KUKA KRL program: redrabbit.src, RedRabbit.dat

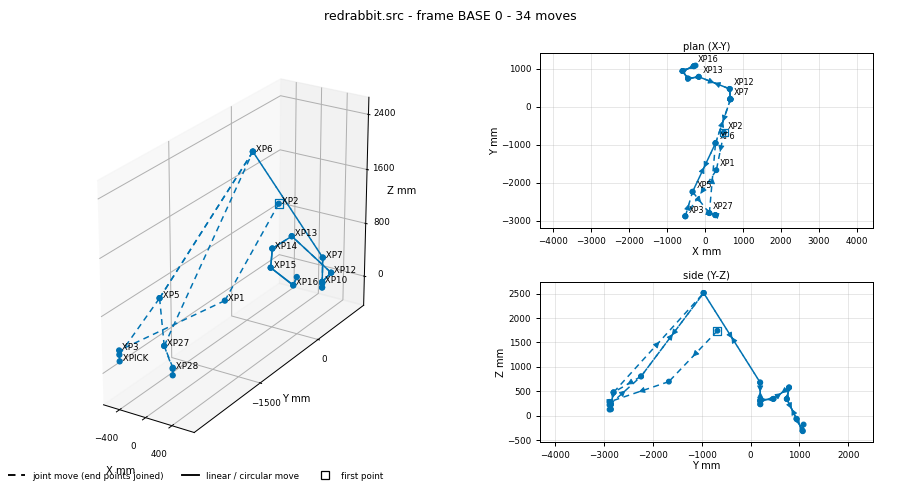
[picture p0: tool path of redrabbit.src in frame BASE 0, 34 of 36 moves have a stored position in this frame; points joined in program order, loops and branches not executed]
--- redrabbit.src ---
&ACCESS RVO1
&REL 74
&PARAM EDITMASK = *
&PARAM TEMPLATE = C:\KRC\TP\Nutweld\Template\NutWeld_Vorgabe
DEF RedRabbit( )
;FOLD INI
  ;FOLD BASISTECH INI
    GLOBAL INTERRUPT DECL 3 WHEN $STOPMESS==TRUE DO IR_STOPM ( )
    INTERRUPT ON 3
    BAS (#INITMOV,0 )
  ;ENDFOLD (BASISTECH INI)
	;FOLD NutWeld
	;ENDFOLD (NutWeld)
  ;FOLD USER INI
    ;Make your modifications here
do141Spare=FALSE
do142Spare=FALSE
  ;ENDFOLD (USER INI)
;ENDFOLD (INI)
wait for false

;FOLD PTP HOME  Vel= 100 % DEFAULT;%{PE}%MKUKATPBASIS,%CMOVE,%VPTP,%P 1:PTP, 2:HOME, 3:, 5:100, 7:DEFAULT
$BWDSTART = FALSE
PDAT_ACT=PDEFAULT
FDAT_ACT=FHOME
BAS (#PTP_PARAMS,100 )
$H_POS=XHOME
PTP  XHOME
;ENDFOLD
;FOLD Gripper SET [1]Gripper1 State=[1]OPEN Wait 0.2[s] Check with Strategy 1 ;%{PE}
;FOLD Parameters Parameters ;%{h}
;Params IlfProvider=GripperTech.GripperSet;setgripper=1;setstate=1;setcont=nocont;waittime=0.2;errorstrategy=1
;ENDFOLD
GRPg_SetStateAndCheck(1, 1, 0.2, 1)
;ENDFOLD
;FOLD Gripper SET [2]Gripper2 State=[2]CLOSE Wait 0.2[s] Check with Strategy 1 ;%{PE}
;FOLD Parameters Parameters ;%{h}
;Params IlfProvider=GripperTech.GripperSet;setgripper=2;setstate=2;setcont=nocont;waittime=0.2;errorstrategy=1
;ENDFOLD
GRPg_SetStateAndCheck(2, 2, 0.2, 1)
;ENDFOLD
;FOLD Gripper SET [3]Gripper3 State=[1]OPEN Wait 0.2[s] Check with Strategy 1 ;%{PE}
;FOLD Parameters Parameters ;%{h}
;Params IlfProvider=GripperTech.GripperSet;setgripper=3;setstate=1;setcont=nocont;waittime=0.2;errorstrategy=1
;ENDFOLD
GRPg_SetStateAndCheck(3, 1, 0.2, 1)
;ENDFOLD
;FOLD Gripper SET [4]Gripper4 State=[2]CLOSE Wait 0.2[s] Check with Strategy 1 ;%{PE}
;FOLD Parameters Parameters ;%{h}
;Params IlfProvider=GripperTech.GripperSet;setgripper=4;setstate=2;setcont=nocont;waittime=0.2;errorstrategy=1
;ENDFOLD
GRPg_SetStateAndCheck(4, 2, 0.2, 1)
;ENDFOLD
;FOLD PTP P2 Vel=100 % PDAT2 Tool[1]:TOOL 1 Base[0];%{PE}%R 8.3.43,%MKUKATPBASIS,%CMOVE,%VPTP,%P 1:PTP, 2:P2, 3:, 5:100, 7:PDAT2
$BWDSTART=FALSE
PDAT_ACT=PPDAT2
FDAT_ACT=FP2
BAS(#PTP_PARAMS,100)
PTP XP2
;ENDFOLD
;FOLD PTP P1 Vel=100 % PDAT1 Tool[1]:TOOL 1 Base[0];%{PE}%R 8.3.43,%MKUKATPBASIS,%CMOVE,%VPTP,%P 1:PTP, 2:P1, 3:, 5:100, 7:PDAT1
$BWDSTART=FALSE
PDAT_ACT=PPDAT1
FDAT_ACT=FP1
BAS(#PTP_PARAMS,100)
PTP XP1
;ENDFOLD
;FOLD PTP P3 Vel=100 % PDAT3 Tool[2]:TOOL 2 Base[0];%{PE}%R 8.3.43,%MKUKATPBASIS,%CMOVE,%VPTP,%P 1:PTP, 2:P3, 3:, 5:100, 7:PDAT3
$BWDSTART=FALSE
PDAT_ACT=PPDAT3
FDAT_ACT=FP3
BAS(#PTP_PARAMS,100)
PTP XP3
;ENDFOLD
;FOLD LIN PICK Vel=1 m/s CPDAT1 Tool[2]:TOOL 2 Base[0];%{PE}%R 8.3.43,%MKUKATPBASIS,%CMOVE,%VLIN,%P 1:LIN, 2:PICK, 3:, 5:1, 7:CPDAT1
$BWDSTART=FALSE
LDAT_ACT=LCPDAT1
FDAT_ACT=FPICK
BAS(#CP_PARAMS,1)
LIN XPICK
;ENDFOLD
;FOLD Gripper SET [3]Gripper3 State=[2]CLOSE Wait 0.2[s] Check with Strategy 1 ;%{PE}
;FOLD Parameters Parameters ;%{h}
;Params IlfProvider=GripperTech.GripperSet;setgripper=3;setstate=2;setcont=nocont;waittime=0.2;errorstrategy=1
;ENDFOLD
GRPg_SetStateAndCheck(3, 2, 0.2, 1)
;ENDFOLD
;FOLD Gripper CHECK [3]Gripper3 State=[2]CLOSE with Strategy 1 ;%{PE}
;FOLD Parameters Parameters ;%{h}
;Params IlfProvider=GripperTech.GripperCheck;setgripper=3;setstate=2;setcont=nocont;checkstrategy=1
;ENDFOLD
GRPg_Check(3, 2, FALSE, 1)
;ENDFOLD
;FOLD LIN P4 Vel=1 m/s CPDAT2 Tool[2]:TOOL 2 Base[0];%{PE}%R 8.3.43,%MKUKATPBASIS,%CMOVE,%VLIN,%P 1:LIN, 2:P4, 3:, 5:1, 7:CPDAT2
$BWDSTART=FALSE
LDAT_ACT=LCPDAT2
FDAT_ACT=FP4
BAS(#CP_PARAMS,1)
LIN XP4
;ENDFOLD
;FOLD PTP P5 Vel=100 % PDAT4 Tool[2]:TOOL 2 Base[0];%{PE}%R 8.3.43,%MKUKATPBASIS,%CMOVE,%VPTP,%P 1:PTP, 2:P5, 3:, 5:100, 7:PDAT4
$BWDSTART=FALSE
PDAT_ACT=PPDAT4
FDAT_ACT=FP5
BAS(#PTP_PARAMS,100)
PTP XP5
;ENDFOLD
;FOLD PTP P6 Vel=100 % PDAT5 Tool[2]:TOOL 2 Base[0];%{PE}%R 8.3.43,%MKUKATPBASIS,%CMOVE,%VPTP,%P 1:PTP, 2:P6, 3:, 5:100, 7:PDAT5
$BWDSTART=FALSE
PDAT_ACT=PPDAT5
FDAT_ACT=FP6
BAS(#PTP_PARAMS,100)
PTP XP6
;ENDFOLD
;Pick RH RedRabbit
;FOLD OUT 120 'do120Spare' State=TRUE ;%{PE}%R 8.3.43,%MKUKATPBASIS,%COUT,%VOUTX,%P 2:120, 3:do120Spare, 5:TRUE, 6:
$OUT[120]=TRUE
;ENDFOLD
;FOLD WAIT FOR ( IN 98 'di098Spare' );%{PE}%R 8.3.43,%MKUKATPBASIS,%CEXT_WAIT_FOR,%VEXT_WAIT_FOR,%P 2:, 4:, 5:$IN, 6:98, 7:di098Spare, 9:
WAIT FOR  ( $IN[98] )
;ENDFOLD
;FOLD PTP P7 Vel=100 % PDAT9 Tool[2]:TOOL 2 Base[0];%{PE}%R 8.3.43,%MKUKATPBASIS,%CMOVE,%VPTP,%P 1:PTP, 2:P7, 3:, 5:100, 7:PDAT9
$BWDSTART=FALSE
PDAT_ACT=PPDAT9
FDAT_ACT=FP7
BAS(#PTP_PARAMS,100)
PTP XP7
;ENDFOLD
;FOLD LIN P10 Vel=1 m/s CPDAT4 Tool[2]:TOOL 2 Base[0];%{PE}%R 8.3.43,%MKUKATPBASIS,%CMOVE,%VLIN,%P 1:LIN, 2:P10, 3:, 5:1, 7:CPDAT4
$BWDSTART=FALSE
LDAT_ACT=LCPDAT4
FDAT_ACT=FP10
BAS(#CP_PARAMS,1)
LIN XP10
;ENDFOLD
;FOLD LIN PICK2 Vel=1 m/s CPDAT5 Tool[2]:TOOL 2 Base[0];%{PE}%R 8.3.43,%MKUKATPBASIS,%CMOVE,%VLIN,%P 1:LIN, 2:PICK2, 3:, 5:1, 7:CPDAT5
$BWDSTART=FALSE
LDAT_ACT=LCPDAT5
FDAT_ACT=FPICK2
BAS(#CP_PARAMS,1)
LIN XPICK2
;ENDFOLD
;FOLD Gripper SET [1]Gripper1 State=[2]CLOSE Wait 0.2[s] Check with Strategy 1 ;%{PE}
;FOLD Parameters Parameters ;%{h}
;Params IlfProvider=GripperTech.GripperSet;setgripper=1;setstate=2;setcont=nocont;waittime=0.2;errorstrategy=1
;ENDFOLD
GRPg_SetStateAndCheck(1, 2, 0.2, 1)
;ENDFOLD
;FOLD Gripper CHECK [1]Gripper1 State=[2]CLOSE with Strategy 1 ;%{PE}
;FOLD Parameters Parameters ;%{h}
;Params IlfProvider=GripperTech.GripperCheck;setgripper=1;setstate=2;setcont=nocont;checkstrategy=1
;ENDFOLD
GRPg_Check(1, 2, FALSE, 1)
;ENDFOLD
;FOLD LIN P11 Vel=1 m/s CPDAT6 Tool[2]:TOOL 2 Base[0];%{PE}%R 8.3.43,%MKUKATPBASIS,%CMOVE,%VLIN,%P 1:LIN, 2:P11, 3:, 5:1, 7:CPDAT6
$BWDSTART=FALSE
LDAT_ACT=LCPDAT6
FDAT_ACT=FP11
BAS(#CP_PARAMS,1)
LIN XP11
;ENDFOLD
;FOLD LIN P12 Vel=1 m/s CPDAT7 Tool[2]:TOOL 2 Base[0];%{PE}%R 8.3.43,%MKUKATPBASIS,%CMOVE,%VLIN,%P 1:LIN, 2:P12, 3:, 5:1, 7:CPDAT7
$BWDSTART=FALSE
LDAT_ACT=LCPDAT7
FDAT_ACT=FP12
BAS(#CP_PARAMS,1)
LIN XP12
;ENDFOLD
;FOLD PTP P13 Vel=100 % PDAT10 Tool[2]:TOOL 2 Base[0];%{PE}%R 8.3.43,%MKUKATPBASIS,%CMOVE,%VPTP,%P 1:PTP, 2:P13, 3:, 5:100, 7:PDAT10
$BWDSTART=FALSE
PDAT_ACT=PPDAT10
FDAT_ACT=FP13
BAS(#PTP_PARAMS,100)
PTP XP13
;ENDFOLD
;FOLD LIN P14 Vel=1 m/s CPDAT8 Tool[2]:TOOL 2 Base[0];%{PE}%R 8.3.43,%MKUKATPBASIS,%CMOVE,%VLIN,%P 1:LIN, 2:P14, 3:, 5:1, 7:CPDAT8
$BWDSTART=FALSE
LDAT_ACT=LCPDAT8
FDAT_ACT=FP14
BAS(#CP_PARAMS,1)
LIN XP14
;ENDFOLD
;FOLD LIN P15 Vel=1 m/s CPDAT9 Tool[2]:TOOL 2 Base[0];%{PE}%R 8.3.43,%MKUKATPBASIS,%CMOVE,%VLIN,%P 1:LIN, 2:P15, 3:, 5:1, 7:CPDAT9
$BWDSTART=FALSE
LDAT_ACT=LCPDAT9
FDAT_ACT=FP15
BAS(#CP_PARAMS,1)
LIN XP15
;ENDFOLD
;FOLD LIN P16 Vel=1 m/s CPDAT10 Tool[2]:TOOL 2 Base[0];%{PE}%R 8.3.43,%MKUKATPBASIS,%CMOVE,%VLIN,%P 1:LIN, 2:P16, 3:, 5:1, 7:CPDAT10
$BWDSTART=FALSE
LDAT_ACT=LCPDAT10
FDAT_ACT=FP16
BAS(#CP_PARAMS,1)
LIN XP16
;ENDFOLD
;FOLD LIN NUTCHECK Vel=1 m/s CPDAT11 Tool[2]:TOOL 2 Base[0];%{PE}%R 8.3.43,%MKUKATPBASIS,%CMOVE,%VLIN,%P 1:LIN, 2:NUTCHECK, 3:, 5:1, 7:CPDAT11
$BWDSTART=FALSE
LDAT_ACT=LCPDAT11
FDAT_ACT=FNUTCHECK
BAS(#CP_PARAMS,1)
LIN XNUTCHECK
;ENDFOLD
;FOLD WAIT Time=1 sec;%{PE}%R 8.3.43,%MKUKATPBASIS,%CWAIT,%VWAIT,%P 3:1
WAIT SEC 1
;ENDFOLD
IF ((di777StudPartPresent1==FALSE) AND (di778StudPartPresent2==FALSE) AND (di779StudPartPresent3==FALSE) AND (di780StudPartPresent4==FALSE) AND (Di781StudPartPresent5==FALSE) AND (di782StudPartPresent6==FALSE)) THEN
do142Spare=TRUE
ELSE
do141Spare=TRUE
ENDIF
;FOLD PTP P17 Vel=100 % PDAT11 Tool[2]:TOOL 2 Base[0];%{PE}%R 8.3.43,%MKUKATPBASIS,%CMOVE,%VPTP,%P 1:PTP, 2:P17, 3:, 5:100, 7:PDAT11
$BWDSTART=FALSE
PDAT_ACT=PPDAT11
FDAT_ACT=FP17
BAS(#PTP_PARAMS,100)
PTP XP17
;ENDFOLD
;FOLD LIN P18 Vel=1 m/s CPDAT12 Tool[2]:TOOL 2 Base[0];%{PE}%R 8.3.43,%MKUKATPBASIS,%CMOVE,%VLIN,%P 1:LIN, 2:P18, 3:, 5:1, 7:CPDAT12
$BWDSTART=FALSE
LDAT_ACT=LCPDAT12
FDAT_ACT=FP18
BAS(#CP_PARAMS,1)
LIN XP18
;ENDFOLD
;FOLD LIN P19 Vel=1 m/s CPDAT13 Tool[2]:TOOL 2 Base[0];%{PE}%R 8.3.43,%MKUKATPBASIS,%CMOVE,%VLIN,%P 1:LIN, 2:P19, 3:, 5:1, 7:CPDAT13
$BWDSTART=FALSE
LDAT_ACT=LCPDAT13
FDAT_ACT=FP19
BAS(#CP_PARAMS,1)
LIN XP19
;ENDFOLD
;FOLD PTP P20 Vel=100 % PDAT12 Tool[2]:TOOL 2 Base[0];%{PE}%R 8.3.43,%MKUKATPBASIS,%CMOVE,%VPTP,%P 1:PTP, 2:P20, 3:, 5:100, 7:PDAT12
$BWDSTART=FALSE
PDAT_ACT=PPDAT12
FDAT_ACT=FP20
BAS(#PTP_PARAMS,100)
PTP XP20
;ENDFOLD
;FOLD LIN P21 Vel=1 m/s CPDAT14 Tool[2]:TOOL 2 Base[0];%{PE}%R 8.3.43,%MKUKATPBASIS,%CMOVE,%VLIN,%P 1:LIN, 2:P21, 3:, 5:1, 7:CPDAT14
$BWDSTART=FALSE
LDAT_ACT=LCPDAT14
FDAT_ACT=FP21
BAS(#CP_PARAMS,1)
LIN XP21
;ENDFOLD
;FOLD LIN P22 Vel=1 m/s CPDAT15 Tool[2]:TOOL 2 Base[0];%{PE}%R 8.3.43,%MKUKATPBASIS,%CMOVE,%VLIN,%P 1:LIN, 2:P22, 3:, 5:1, 7:CPDAT15
$BWDSTART=FALSE
LDAT_ACT=LCPDAT15
FDAT_ACT=FP22
BAS(#CP_PARAMS,1)
LIN XP22
;ENDFOLD
;FOLD LIN DROP Vel=1 m/s CPDAT16 Tool[2]:TOOL 2 Base[0];%{PE}%R 8.3.43,%MKUKATPBASIS,%CMOVE,%VLIN,%P 1:LIN, 2:DROP, 3:, 5:1, 7:CPDAT16
$BWDSTART=FALSE
LDAT_ACT=LCPDAT16
FDAT_ACT=FDROP
BAS(#CP_PARAMS,1)
LIN XDROP
;ENDFOLD
;FOLD Gripper SET [2]Gripper2 State=[1]OPEN Wait 0.2[s] Check with Strategy 1 ;%{PE}
;FOLD Parameters Parameters ;%{h}
;Params IlfProvider=GripperTech.GripperSet;setgripper=2;setstate=1;setcont=nocont;waittime=0.2;errorstrategy=1
;ENDFOLD
GRPg_SetStateAndCheck(2, 1, 0.2, 1)
;ENDFOLD
;FOLD Gripper SET [1]Gripper1 State=[1]OPEN Wait 0.2[s] Check with Strategy 1 ;%{PE}
;FOLD Parameters Parameters ;%{h}
;Params IlfProvider=GripperTech.GripperSet;setgripper=1;setstate=1;setcont=nocont;waittime=0.2;errorstrategy=1
;ENDFOLD
GRPg_SetStateAndCheck(1, 1, 0.2, 1)
;ENDFOLD
;FOLD Gripper CHECK [2]Gripper2 State=[1]OPEN with Strategy 1 ;%{PE}
;FOLD Parameters Parameters ;%{h}
;Params IlfProvider=GripperTech.GripperCheck;setgripper=2;setstate=1;setcont=nocont;checkstrategy=1
;ENDFOLD
GRPg_Check(2, 1, FALSE, 1)
;ENDFOLD
;FOLD Gripper CHECK [1]Gripper1 State=[1]OPEN with Strategy 1 ;%{PE}
;FOLD Parameters Parameters ;%{h}
;Params IlfProvider=GripperTech.GripperCheck;setgripper=1;setstate=1;setcont=nocont;checkstrategy=1
;ENDFOLD
GRPg_Check(1, 1, FALSE, 1)
;ENDFOLD
;FOLD LIN P23 Vel=1 m/s CPDAT17 Tool[2]:TOOL 2 Base[0];%{PE}%R 8.3.43,%MKUKATPBASIS,%CMOVE,%VLIN,%P 1:LIN, 2:P23, 3:, 5:1, 7:CPDAT17
$BWDSTART=FALSE
LDAT_ACT=LCPDAT17
FDAT_ACT=FP23
BAS(#CP_PARAMS,1)
LIN XP23
;ENDFOLD
;FOLD PTP P24 Vel=100 % PDAT13 Tool[2]:TOOL 2 Base[0];%{PE}%R 8.3.43,%MKUKATPBASIS,%CMOVE,%VPTP,%P 1:PTP, 2:P24, 3:, 5:100, 7:PDAT13
$BWDSTART=FALSE
PDAT_ACT=PPDAT13
FDAT_ACT=FP24
BAS(#PTP_PARAMS,100)
PTP XP24
;ENDFOLD
;FOLD PTP P25 Vel=100 % PDAT14 Tool[2]:TOOL 2 Base[0];%{PE}%R 8.3.43,%MKUKATPBASIS,%CMOVE,%VPTP,%P 1:PTP, 2:P25, 3:, 5:100, 7:PDAT14
$BWDSTART=FALSE
PDAT_ACT=PPDAT14
FDAT_ACT=FP25
BAS(#PTP_PARAMS,100)
PTP XP25
;ENDFOLD
;FOLD OUT 120 'do120Spare' State=FALSE ;%{PE}%R 8.3.43,%MKUKATPBASIS,%COUT,%VOUTX,%P 2:120, 3:do120Spare, 5:FALSE, 6:
$OUT[120]=FALSE
;ENDFOLD
;FOLD PTP P26 Vel=100 % PDAT15 Tool[2]:TOOL 2 Base[0];%{PE}%R 8.3.43,%MKUKATPBASIS,%CMOVE,%VPTP,%P 1:PTP, 2:P26, 3:, 5:100, 7:PDAT15
$BWDSTART=FALSE
PDAT_ACT=PPDAT15
FDAT_ACT=FP26
BAS(#PTP_PARAMS,100)
PTP XP26
;ENDFOLD
;FOLD PTP P27 Vel=100 % PDAT16 Tool[2]:TOOL 2 Base[0];%{PE}%R 8.3.43,%MKUKATPBASIS,%CMOVE,%VPTP,%P 1:PTP, 2:P27, 3:, 5:100, 7:PDAT16
$BWDSTART=FALSE
PDAT_ACT=PPDAT16
FDAT_ACT=FP27
BAS(#PTP_PARAMS,100)
PTP XP27
;ENDFOLD
;FOLD PTP P28 Vel=100 % PDAT17 Tool[2]:TOOL 2 Base[0];%{PE}%R 8.3.43,%MKUKATPBASIS,%CMOVE,%VPTP,%P 1:PTP, 2:P28, 3:, 5:100, 7:PDAT17
$BWDSTART=FALSE
PDAT_ACT=PPDAT17
FDAT_ACT=FP28
BAS(#PTP_PARAMS,100)
PTP XP28
;ENDFOLD
;FOLD LIN DROP2 Vel=1 m/s CPDAT18 Tool[2]:TOOL 2 Base[0];%{PE}%R 8.3.43,%MKUKATPBASIS,%CMOVE,%VLIN,%P 1:LIN, 2:DROP2, 3:, 5:1, 7:CPDAT18
$BWDSTART=FALSE
LDAT_ACT=LCPDAT18
FDAT_ACT=FDROP2
BAS(#CP_PARAMS,1)
LIN XDROP2
;ENDFOLD
;FOLD Gripper SET [3]Gripper3 State=[1]OPEN Wait 0.2[s] Check with Strategy 1 ;%{PE}
;FOLD Parameters Parameters ;%{h}
;Params IlfProvider=GripperTech.GripperSet;setgripper=3;setstate=1;setcont=nocont;waittime=0.2;errorstrategy=1
;ENDFOLD
GRPg_SetStateAndCheck(3, 1, 0.2, 1)
;ENDFOLD
;FOLD Gripper CHECK [3]Gripper3 State=[1]OPEN with Strategy 1 ;%{PE}
;FOLD Parameters Parameters ;%{h}
;Params IlfProvider=GripperTech.GripperCheck;setgripper=3;setstate=1;setcont=nocont;checkstrategy=1
;ENDFOLD
GRPg_Check(3, 1, FALSE, 1)
;ENDFOLD
;FOLD LIN P29 Vel=1 m/s CPDAT19 Tool[2]:TOOL 2 Base[0];%{PE}%R 8.3.43,%MKUKATPBASIS,%CMOVE,%VLIN,%P 1:LIN, 2:P29, 3:, 5:1, 7:CPDAT19
$BWDSTART=FALSE
LDAT_ACT=LCPDAT19
FDAT_ACT=FP29
BAS(#CP_PARAMS,1)
LIN XP29
;ENDFOLD
;FOLD PTP P30 Vel=100 % PDAT18 Tool[2]:TOOL 2 Base[0];%{PE}%R 8.3.43,%MKUKATPBASIS,%CMOVE,%VPTP,%P 1:PTP, 2:P30, 3:, 5:100, 7:PDAT18
$BWDSTART=FALSE
PDAT_ACT=PPDAT18
FDAT_ACT=FP30
BAS(#PTP_PARAMS,100)
PTP XP30
;ENDFOLD
;FOLD PTP P31 Vel=100 % PDAT19 Tool[2]:TOOL 2 Base[0];%{PE}%R 8.3.43,%MKUKATPBASIS,%CMOVE,%VPTP,%P 1:PTP, 2:P31, 3:, 5:100, 7:PDAT19
$BWDSTART=FALSE
PDAT_ACT=PPDAT19
FDAT_ACT=FP31
BAS(#PTP_PARAMS,100)
PTP XP31
;ENDFOLD
;FOLD PTP HOME  Vel= 100 % DEFAULT;%{PE}%MKUKATPBASIS,%CMOVE,%VPTP,%P 1:PTP, 2:HOME, 3:, 5:100, 7:DEFAULT
$BWDSTART = FALSE
PDAT_ACT=PDEFAULT
FDAT_ACT=FHOME
BAS (#PTP_PARAMS,100 )
$H_POS=XHOME
PTP  XHOME
;ENDFOLD

END

--- RedRabbit.dat ---
&ACCESS RVO1
&REL 74
&PARAM EDITMASK = *
&PARAM TEMPLATE = C:\KRC\TP\Nutweld\Template\NutWeld_Vorgabe
DEFDAT  RedRabbit
;FOLD EXTERNAL DECLARATIONS;%{PE}%MKUKATPBASIS,%CEXT,%VCOMMON,%P
;FOLD BASISTECH EXT;%{PE}%MKUKATPBASIS,%CEXT,%VEXT,%P
EXT  BAS (BAS_COMMAND  :IN,REAL  :IN )
DECL INT SUCCESS
;ENDFOLD (BASISTECH EXT)
;FOLD NutWeld
BOOL NutWeld_TEMPLATE=TRUE
;ENDFOLD (NutWeld)
;FOLD USER EXT;%{E}%MKUKATPUSER,%CEXT,%VEXT,%P
;Make here your modifications

;ENDFOLD (USER EXT)
;ENDFOLD (EXTERNAL DECLARATIONS)
DECL BASIS_SUGG_T LAST_BASIS={POINT1[] "P31                     ",POINT2[] "P31                     ",CP_PARAMS[] "CPDAT19                 ",PTP_PARAMS[] "PDAT19                  ",CONT[] "                        ",CP_VEL[] "1                       ",PTP_VEL[] "100                     ",SYNC_PARAMS[] "SYNCDAT                 ",SPL_NAME[] "S0                      ",A_PARAMS[] "ADAT0                   "}
DECL E6POS XP1={X 300.792389,Y -1670.96313,Z 699.152344,A 1.40872371,B -0.137058839,C -178.656876,S 2,T 42,E1 0.0,E2 0.0,E3 0.0,E4 0.0,E5 0.0,E6 0.0}
DECL FDAT FP1={TOOL_NO 1,BASE_NO 0,IPO_FRAME #BASE,POINT2[] " ",TQ_STATE FALSE}
DECL PDAT PPDAT1={VEL 100.000,ACC 100.000,APO_DIST 100.000,APO_MODE #CDIS,GEAR_JERK 50.0000,EXAX_IGN 0}
DECL E6POS XP2={X 501.960907,Y -678.097229,Z 1739.82629,A 27.3295097,B 26.7028427,C 117.650810,S 2,T 42,E1 0.0,E2 0.0,E3 0.0,E4 0.0,E5 0.0,E6 0.0}
DECL FDAT FP2={TOOL_NO 1,BASE_NO 0,IPO_FRAME #BASE,POINT2[] " ",TQ_STATE FALSE}
DECL PDAT PPDAT2={VEL 100.000,ACC 100.000,APO_DIST 100.000,APO_MODE #CDIS,GEAR_JERK 50.0000,EXAX_IGN 0}
DECL E6POS XPICK={X -515.437317,Y -2883.09497,Z 127.622879,A -82.2796097,B 1.14908242,C -179.579742,S 2,T 42,E1 0.0,E2 0.0,E3 0.0,E4 0.0,E5 0.0,E6 0.0}
DECL FDAT FPICK={TOOL_NO 2,BASE_NO 0,IPO_FRAME #BASE,POINT2[] " ",TQ_STATE FALSE}
DECL LDAT LCPDAT1={VEL 2.00000,ACC 100.000,APO_DIST 100.000,APO_FAC 50.0000,AXIS_VEL 100.000,AXIS_ACC 100.000,ORI_TYP #VAR,CIRC_TYP #BASE,JERK_FAC 50.0000,GEAR_JERK 50.0000,EXAX_IGN 0}
DECL E6POS XP3={X -516.039429,Y -2887.24805,Z 284.975098,A -81.9615784,B 1.46866310,C -179.571594,S 2,T 34,E1 0.0,E2 0.0,E3 0.0,E4 0.0,E5 0.0,E6 0.0}
DECL FDAT FP3={TOOL_NO 2,BASE_NO 0,IPO_FRAME #BASE,POINT2[] " ",TQ_STATE FALSE}
DECL PDAT PPDAT3={VEL 100.000,ACC 100.000,APO_DIST 100.000,APO_MODE #CDIS,GEAR_JERK 50.0000,EXAX_IGN 0}
DECL E6POS XP4={X -515.872070,Y -2885.07715,Z 222.640778,A -82.2796097,B 1.14908242,C -179.579742,S 2,T 42,E1 0.0,E2 0.0,E3 0.0,E4 0.0,E5 0.0,E6 0.0}
DECL FDAT FP4={TOOL_NO 2,BASE_NO 0,IPO_FRAME #BASE,POINT2[] " ",TQ_STATE FALSE}
DECL LDAT LCPDAT2={VEL 2.00000,ACC 100.000,APO_DIST 100.000,APO_FAC 50.0000,AXIS_VEL 100.000,AXIS_ACC 100.000,ORI_TYP #VAR,CIRC_TYP #BASE,JERK_FAC 50.0000,GEAR_JERK 50.0000,EXAX_IGN 0}
DECL E6POS XP5={X -325.126160,Y -2239.52100,Z 805.829956,A -88.5880661,B 1.34312057,C -179.862900,S 2,T 42,E1 0.0,E2 0.0,E3 0.0,E4 0.0,E5 0.0,E6 0.0}
DECL FDAT FP5={TOOL_NO 2,BASE_NO 0,IPO_FRAME #BASE,POINT2[] " ",TQ_STATE FALSE}
DECL PDAT PPDAT4={VEL 100.000,ACC 100.000,APO_DIST 100.000,APO_MODE #CDIS,GEAR_JERK 50.0000,EXAX_IGN 0}
DECL E6POS XP6={X 279.497772,Y -959.753845,Z 2512.86719,A -22.0508213,B -52.3092079,C 132.694931,S 2,T 42,E1 0.0,E2 0.0,E3 0.0,E4 0.0,E5 0.0,E6 0.0}
DECL FDAT FP6={TOOL_NO 2,BASE_NO 0,IPO_FRAME #BASE,POINT2[] " ",TQ_STATE FALSE}
DECL PDAT PPDAT5={VEL 100.000,ACC 100.000,APO_DIST 100.000,APO_MODE #CDIS,GEAR_JERK 50.0000,EXAX_IGN 0}
DECL E6POS XP7={X 673.698486,Y 196.744370,Z 680.549194,A 179.410934,B 0.188110352,C 179.999451,S 2,T 34,E1 0.0,E2 0.0,E3 0.0,E4 0.0,E5 0.0,E6 0.0}
DECL FDAT FP7={TOOL_NO 2,BASE_NO 0,IPO_FRAME #BASE,POINT2[] " ",TQ_STATE FALSE}
DECL PDAT PPDAT6={VEL 100.000,ACC 100.000,APO_DIST 100.000,APO_MODE #CDIS,GEAR_JERK 50.0000,EXAX_IGN 0}
DECL E6POS XP8={X -121.469971,Y 786.551758,Z 872.609436,A -29.0992374,B 0.730682194,C -179.183685,S 2,T 3,E1 0.0,E2 0.0,E3 0.0,E4 0.0,E5 0.0,E6 0.0}
DECL FDAT FP8={TOOL_NO 2,BASE_NO 0,IPO_FRAME #BASE,POINT2[] " ",TQ_STATE FALSE}
DECL PDAT PPDAT7={VEL 100.000,ACC 100.000,APO_DIST 100.000,APO_MODE #CDIS,GEAR_JERK 50.0000,EXAX_IGN 0}
DECL E6POS XP9={X -283.548,Y 885.343506,Z 348.627655,A -29.0992374,B 0.730682194,C -179.183685,S 2,T 3,E1 0.0,E2 0.0,E3 0.0,E4 0.0,E5 0.0,E6 0.0}
DECL FDAT FP9={TOOL_NO 2,BASE_NO 0,IPO_FRAME #BASE,POINT2[] " ",TQ_STATE FALSE}
DECL PDAT PPDAT8={VEL 100.000,ACC 100.000,APO_DIST 100.000,APO_MODE #CDIS,GEAR_JERK 50.0000,EXAX_IGN 0}
DECL E6POS XNUTCHECK={X -246.798584,Y 1084.69397,Z -178.875153,A -20.3971767,B -0.394200563,C -179.586792,S 2,T 3,E1 0.0,E2 0.0,E3 0.0,E4 0.0,E5 0.0,E6 0.0}
DECL FDAT FNUTCHECK={TOOL_NO 2,BASE_NO 0,IPO_FRAME #BASE,POINT2[] " ",TQ_STATE FALSE}
DECL LDAT LCPDAT3={VEL 2.00000,ACC 100.000,APO_DIST 100.000,APO_FAC 50.0000,AXIS_VEL 100.000,AXIS_ACC 100.000,ORI_TYP #VAR,CIRC_TYP #BASE,JERK_FAC 50.0000,GEAR_JERK 50.0000,EXAX_IGN 0}
DECL PDAT PPDAT9={VEL 100.000,ACC 100.000,APO_DIST 100.000,APO_MODE #CDIS,GEAR_JERK 50.0000,EXAX_IGN 0}
DECL E6POS XP10={X 670.338440,Y 198.063278,Z 299.317383,A 179.574432,B 0.398581892,C -179.632553,S 2,T 35,E1 0.0,E2 0.0,E3 0.0,E4 0.0,E5 0.0,E6 0.0}
DECL FDAT FP10={TOOL_NO 2,BASE_NO 0,IPO_FRAME #BASE,POINT2[] " ",TQ_STATE FALSE}
DECL LDAT LCPDAT4={VEL 2.00000,ACC 100.000,APO_DIST 100.000,APO_FAC 50.0000,AXIS_VEL 100.000,AXIS_ACC 100.000,ORI_TYP #VAR,CIRC_TYP #BASE,JERK_FAC 50.0000,GEAR_JERK 50.0000,EXAX_IGN 0}
DECL E6POS XPICK2={X 669.738403,Y 199.126968,Z 236.324707,A 179.574432,B 0.398581892,C -179.632553,S 2,T 35,E1 0.0,E2 0.0,E3 0.0,E4 0.0,E5 0.0,E6 0.0}
DECL FDAT FPICK2={TOOL_NO 2,BASE_NO 0,IPO_FRAME #BASE,POINT2[] " ",TQ_STATE FALSE}
DECL LDAT LCPDAT5={VEL 2.00000,ACC 100.000,APO_DIST 100.000,APO_FAC 50.0000,AXIS_VEL 100.000,AXIS_ACC 100.000,ORI_TYP #VAR,CIRC_TYP #BASE,JERK_FAC 50.0000,GEAR_JERK 50.0000,EXAX_IGN 0}
DECL E6POS XP11={X 669.164246,Y 199.664261,Z 319.434753,A 179.574432,B 0.398581922,C -179.632553,S 2,T 35,E1 0.0,E2 0.0,E3 0.0,E4 0.0,E5 0.0,E6 0.0}
DECL FDAT FP11={TOOL_NO 2,BASE_NO 0,IPO_FRAME #BASE,POINT2[] " ",TQ_STATE FALSE}
DECL LDAT LCPDAT6={VEL 2.00000,ACC 100.000,APO_DIST 100.000,APO_FAC 50.0000,AXIS_VEL 100.000,AXIS_ACC 100.000,ORI_TYP #VAR,CIRC_TYP #BASE,JERK_FAC 50.0000,GEAR_JERK 50.0000,EXAX_IGN 0}
DECL E6POS XP12={X 653.629578,Y 468.717438,Z 346.617554,A 179.502716,B 0.349512577,C -179.673172,S 2,T 35,E1 0.0,E2 0.0,E3 0.0,E4 0.0,E5 0.0,E6 0.0}
DECL FDAT FP12={TOOL_NO 2,BASE_NO 0,IPO_FRAME #BASE,POINT2[] " ",TQ_STATE FALSE}
DECL LDAT LCPDAT7={VEL 2.00000,ACC 100.000,APO_DIST 100.000,APO_FAC 50.0000,AXIS_VEL 100.000,AXIS_ACC 100.000,ORI_TYP #VAR,CIRC_TYP #BASE,JERK_FAC 50.0000,GEAR_JERK 50.0000,EXAX_IGN 0}
DECL E6POS XP13={X -160.967514,Y 787.468079,Z 579.882507,A -13.1324120,B 8.71148872,C 169.351303,S 2,T 11,E1 0.0,E2 0.0,E3 0.0,E4 0.0,E5 0.0,E6 0.0}
DECL FDAT FP13={TOOL_NO 2,BASE_NO 0,IPO_FRAME #BASE,POINT2[] " ",TQ_STATE FALSE}
DECL PDAT PPDAT10={VEL 100.000,ACC 100.000,APO_DIST 100.000,APO_MODE #CDIS,GEAR_JERK 50.0000,EXAX_IGN 0}
DECL E6POS XP14={X -446.019897,Y 741.696,Z 343.617859,A -37.4753647,B 2.69103980,C 161.369522,S 2,T 11,E1 0.0,E2 0.0,E3 0.0,E4 0.0,E5 0.0,E6 0.0}
DECL FDAT FP14={TOOL_NO 2,BASE_NO 0,IPO_FRAME #BASE,POINT2[] " ",TQ_STATE FALSE}
DECL LDAT LCPDAT8={VEL 2.00000,ACC 100.000,APO_DIST 100.000,APO_FAC 50.0000,AXIS_VEL 100.000,AXIS_ACC 100.000,ORI_TYP #VAR,CIRC_TYP #BASE,JERK_FAC 50.0000,GEAR_JERK 50.0000,EXAX_IGN 0}
DECL E6POS XP15={X -589.916687,Y 939.421387,Z -61.4160614,A -35.3626556,B 2.65734100,C 161.405655,S 2,T 11,E1 0.0,E2 0.0,E3 0.0,E4 0.0,E5 0.0,E6 0.0}
DECL FDAT FP15={TOOL_NO 2,BASE_NO 0,IPO_FRAME #BASE,POINT2[] " ",TQ_STATE FALSE}
DECL LDAT LCPDAT9={VEL 2.00000,ACC 100.000,APO_DIST 100.000,APO_FAC 50.0000,AXIS_VEL 100.000,AXIS_ACC 100.000,ORI_TYP #VAR,CIRC_TYP #BASE,JERK_FAC 50.0000,GEAR_JERK 50.0000,EXAX_IGN 0}
DECL E6POS XP16={X -292.407745,Y 1066.61353,Z -307.441284,A -24.1853428,B -0.223531142,C 178.907654,S 2,T 11,E1 0.0,E2 0.0,E3 0.0,E4 0.0,E5 0.0,E6 0.0}
DECL FDAT FP16={TOOL_NO 2,BASE_NO 0,IPO_FRAME #BASE,POINT2[] " ",TQ_STATE FALSE}
DECL LDAT LCPDAT10={VEL 2.00000,ACC 100.000,APO_DIST 100.000,APO_FAC 50.0000,AXIS_VEL 100.000,AXIS_ACC 100.000,ORI_TYP #VAR,CIRC_TYP #BASE,JERK_FAC 50.0000,GEAR_JERK 50.0000,EXAX_IGN 0}
DECL LDAT LCPDAT11={VEL 2.00000,ACC 100.000,APO_DIST 100.000,APO_FAC 50.0000,AXIS_VEL 100.000,AXIS_ACC 100.000,ORI_TYP #VAR,CIRC_TYP #BASE,JERK_FAC 50.0000,GEAR_JERK 50.0000,EXAX_IGN 0}
DECL E6POS XP17={X -292.400604,Y 1066.59790,Z -315.094269,A -24.1853580,B -0.223589614,C 178.907730,S 2,T 11,E1 0.0,E2 0.0,E3 0.0,E4 0.0,E5 0.0,E6 0.0}
DECL FDAT FP17={TOOL_NO 2,BASE_NO 0,IPO_FRAME #BASE,POINT2[] " ",TQ_STATE FALSE}
DECL PDAT PPDAT11={VEL 100.000,ACC 100.000,APO_DIST 100.000,APO_MODE #CDIS,GEAR_JERK 50.0000,EXAX_IGN 0}
DECL E6POS XP18={X -589.916687,Y 939.421387,Z -61.4160614,A -35.3626556,B 2.65734100,C 161.405655,S 2,T 11,E1 0.0,E2 0.0,E3 0.0,E4 0.0,E5 0.0,E6 0.0}
DECL FDAT FP18={TOOL_NO 2,BASE_NO 0,IPO_FRAME #BASE,POINT2[] " ",TQ_STATE FALSE}
DECL LDAT LCPDAT12={VEL 2.00000,ACC 100.000,APO_DIST 100.000,APO_FAC 50.0000,AXIS_VEL 100.000,AXIS_ACC 100.000,ORI_TYP #VAR,CIRC_TYP #BASE,JERK_FAC 50.0000,GEAR_JERK 50.0000,EXAX_IGN 0}
DECL E6POS XP19={X -446.019897,Y 741.696,Z 343.617859,A -37.4753647,B 2.69103980,C 161.369522,S 2,T 11,E1 0.0,E2 0.0,E3 0.0,E4 0.0,E5 0.0,E6 0.0}
DECL FDAT FP19={TOOL_NO 2,BASE_NO 0,IPO_FRAME #BASE,POINT2[] " ",TQ_STATE FALSE}
DECL LDAT LCPDAT13={VEL 2.00000,ACC 100.000,APO_DIST 100.000,APO_FAC 50.0000,AXIS_VEL 100.000,AXIS_ACC 100.000,ORI_TYP #VAR,CIRC_TYP #BASE,JERK_FAC 50.0000,GEAR_JERK 50.0000,EXAX_IGN 0}
DECL E6POS XP20={X -160.967514,Y 787.468079,Z 579.882507,A -13.1324120,B 8.71148872,C 169.351303,S 2,T 11,E1 0.0,E2 0.0,E3 0.0,E4 0.0,E5 0.0,E6 0.0}
DECL FDAT FP20={TOOL_NO 2,BASE_NO 0,IPO_FRAME #BASE,POINT2[] " ",TQ_STATE FALSE}
DECL PDAT PPDAT12={VEL 100.000,ACC 100.000,APO_DIST 100.000,APO_MODE #CDIS,GEAR_JERK 50.0000,EXAX_IGN 0}
DECL E6POS XP21={X 653.629578,Y 468.717438,Z 346.617554,A 179.502716,B 0.349512577,C -179.673172,S 2,T 35,E1 0.0,E2 0.0,E3 0.0,E4 0.0,E5 0.0,E6 0.0}
DECL FDAT FP21={TOOL_NO 2,BASE_NO 0,IPO_FRAME #BASE,POINT2[] " ",TQ_STATE FALSE}
DECL LDAT LCPDAT14={VEL 2.00000,ACC 100.000,APO_DIST 100.000,APO_FAC 50.0000,AXIS_VEL 100.000,AXIS_ACC 100.000,ORI_TYP #VAR,CIRC_TYP #BASE,JERK_FAC 50.0000,GEAR_JERK 50.0000,EXAX_IGN 0}
DECL E6POS XP22={X 669.164246,Y 199.664261,Z 319.434753,A 179.574432,B 0.398581922,C -179.632553,S 2,T 35,E1 0.0,E2 0.0,E3 0.0,E4 0.0,E5 0.0,E6 0.0}
DECL FDAT FP22={TOOL_NO 2,BASE_NO 0,IPO_FRAME #BASE,POINT2[] " ",TQ_STATE FALSE}
DECL LDAT LCPDAT15={VEL 2.00000,ACC 100.000,APO_DIST 100.000,APO_FAC 50.0000,AXIS_VEL 100.000,AXIS_ACC 100.000,ORI_TYP #VAR,CIRC_TYP #BASE,JERK_FAC 50.0000,GEAR_JERK 50.0000,EXAX_IGN 0}
DECL E6POS XDROP={X 669.738403,Y 199.126968,Z 236.324707,A 179.574432,B 0.398581922,C -179.632553,S 2,T 35,E1 0.0,E2 0.0,E3 0.0,E4 0.0,E5 0.0,E6 0.0}
DECL FDAT FDROP={TOOL_NO 2,BASE_NO 0,IPO_FRAME #BASE,POINT2[] " ",TQ_STATE FALSE}
DECL LDAT LCPDAT16={VEL 2.00000,ACC 100.000,APO_DIST 100.000,APO_FAC 50.0000,AXIS_VEL 100.000,AXIS_ACC 100.000,ORI_TYP #VAR,CIRC_TYP #BASE,JERK_FAC 50.0000,GEAR_JERK 50.0000,EXAX_IGN 0}
DECL E6POS XP23={X 670.338440,Y 198.063278,Z 299.317383,A 179.574432,B 0.398581922,C -179.632553,S 2,T 35,E1 0.0,E2 0.0,E3 0.0,E4 0.0,E5 0.0,E6 0.0}
DECL FDAT FP23={TOOL_NO 2,BASE_NO 0,IPO_FRAME #BASE,POINT2[] " ",TQ_STATE FALSE}
DECL LDAT LCPDAT17={VEL 2.00000,ACC 100.000,APO_DIST 100.000,APO_FAC 50.0000,AXIS_VEL 100.000,AXIS_ACC 100.000,ORI_TYP #VAR,CIRC_TYP #BASE,JERK_FAC 50.0000,GEAR_JERK 50.0000,EXAX_IGN 0}
DECL E6POS XP24={X 673.698425,Y 196.744370,Z 680.549194,A 179.410934,B 0.188111514,C 179.999451,S 2,T 34,E1 0.0,E2 0.0,E3 0.0,E4 0.0,E5 0.0,E6 0.0}
DECL FDAT FP24={TOOL_NO 2,BASE_NO 0,IPO_FRAME #BASE,POINT2[] " ",TQ_STATE FALSE}
DECL PDAT PPDAT13={VEL 100.000,ACC 100.000,APO_DIST 100.000,APO_MODE #CDIS,GEAR_JERK 50.0000,EXAX_IGN 0}
DECL E6POS XP25={X 279.497772,Y -959.753845,Z 2512.86719,A -22.0508213,B -52.3092079,C 132.694931,S 2,T 42,E1 0.0,E2 0.0,E3 0.0,E4 0.0,E5 0.0,E6 0.0}
DECL FDAT FP25={TOOL_NO 2,BASE_NO 0,IPO_FRAME #BASE,POINT2[] " ",TQ_STATE FALSE}
DECL PDAT PPDAT14={VEL 100.000,ACC 100.000,APO_DIST 100.000,APO_MODE #CDIS,GEAR_JERK 50.0000,EXAX_IGN 0}
DECL E6POS XP26={X -325.126160,Y -2239.52100,Z 805.829956,A -88.5880661,B 1.34312057,C -179.862900,S 2,T 42,E1 0.0,E2 0.0,E3 0.0,E4 0.0,E5 0.0,E6 0.0}
DECL FDAT FP26={TOOL_NO 2,BASE_NO 0,IPO_FRAME #BASE,POINT2[] " ",TQ_STATE FALSE}
DECL PDAT PPDAT15={VEL 100.000,ACC 100.000,APO_DIST 100.000,APO_MODE #CDIS,GEAR_JERK 50.0000,EXAX_IGN 0}
DECL E6POS XP27={X 116.934715,Y -2801.87329,Z 480.235840,A -39.3507195,B 0.773205101,C -178.893204,S 2,T 42,E1 0.0,E2 0.0,E3 0.0,E4 0.0,E5 0.0,E6 0.0}
DECL FDAT FP27={TOOL_NO 2,BASE_NO 0,IPO_FRAME #BASE,POINT2[] " ",TQ_STATE FALSE}
DECL PDAT PPDAT16={VEL 100.000,ACC 100.000,APO_DIST 100.000,APO_MODE #CDIS,GEAR_JERK 50.0000,EXAX_IGN 0}
DECL E6POS XP28={X 275.960144,Y -2857.37451,Z 227.064957,A -42.7928925,B 0.400950789,C -179.811920,S 2,T 34,E1 0.0,E2 0.0,E3 0.0,E4 0.0,E5 0.0,E6 0.0}
DECL FDAT FP28={TOOL_NO 2,BASE_NO 0,IPO_FRAME #BASE,POINT2[] " ",TQ_STATE FALSE}
DECL PDAT PPDAT17={VEL 100.000,ACC 100.000,APO_DIST 100.000,APO_MODE #CDIS,GEAR_JERK 50.0000,EXAX_IGN 0}
DECL E6POS XDROP2={X 274.714478,Y -2854.79810,Z 132.557800,A -42.6780205,B 0.400061935,C 178.558731,S 2,T 34,E1 0.0,E2 0.0,E3 0.0,E4 0.0,E5 0.0,E6 0.0}
DECL FDAT FDROP2={TOOL_NO 2,BASE_NO 0,IPO_FRAME #BASE,POINT2[] " ",TQ_STATE FALSE}
DECL LDAT LCPDAT18={VEL 2.00000,ACC 100.000,APO_DIST 100.000,APO_FAC 50.0000,AXIS_VEL 100.000,AXIS_ACC 100.000,ORI_TYP #VAR,CIRC_TYP #BASE,JERK_FAC 50.0000,GEAR_JERK 50.0000,EXAX_IGN 0}
DECL E6POS XP29={X 277.071228,Y -2853.33618,Z 238.768326,A -42.6780205,B 0.400061905,C 178.558731,S 2,T 34,E1 0.0,E2 0.0,E3 0.0,E4 0.0,E5 0.0,E6 0.0}
DECL FDAT FP29={TOOL_NO 2,BASE_NO 0,IPO_FRAME #BASE,POINT2[] " ",TQ_STATE FALSE}
DECL LDAT LCPDAT19={VEL 2.00000,ACC 100.000,APO_DIST 100.000,APO_FAC 50.0000,AXIS_VEL 100.000,AXIS_ACC 100.000,ORI_TYP #VAR,CIRC_TYP #BASE,JERK_FAC 50.0000,GEAR_JERK 50.0000,EXAX_IGN 0}
DECL E6POS XP30={X 116.934799,Y -2801.87329,Z 480.235840,A -39.3507195,B 0.773206592,C -178.893204,S 2,T 42,E1 0.0,E2 0.0,E3 0.0,E4 0.0,E5 0.0,E6 0.0}
DECL FDAT FP30={TOOL_NO 2,BASE_NO 0,IPO_FRAME #BASE,POINT2[] " ",TQ_STATE FALSE}
DECL PDAT PPDAT18={VEL 100.000,ACC 100.000,APO_DIST 100.000,APO_MODE #CDIS,GEAR_JERK 50.0000,EXAX_IGN 0}
DECL E6POS XP31={X 279.497772,Y -959.753845,Z 2512.86719,A -22.0508213,B -52.3092079,C 132.694931,S 2,T 42,E1 0.0,E2 0.0,E3 0.0,E4 0.0,E5 0.0,E6 0.0}
DECL FDAT FP31={TOOL_NO 2,BASE_NO 0,IPO_FRAME #BASE,POINT2[] " ",TQ_STATE FALSE}
DECL PDAT PPDAT19={VEL 100.000,ACC 100.000,APO_DIST 100.000,APO_MODE #CDIS,GEAR_JERK 50.0000,EXAX_IGN 0}
ENDDAT
